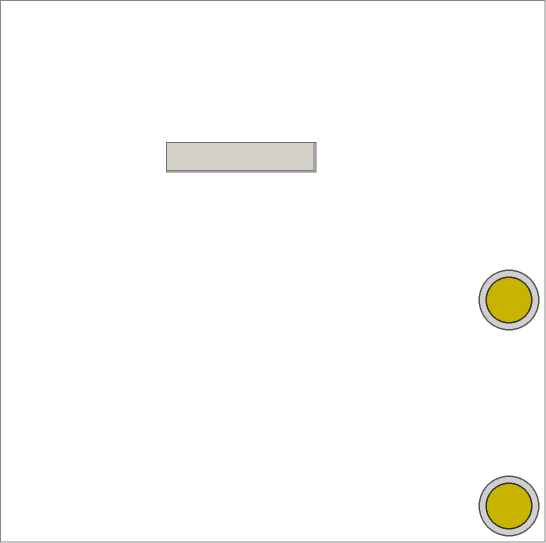
VISUALIZATION Visualization  // 546x543
    Button (166,142 150x30)
        OnMouseClick: toggle MAIN.inputValue
        OnMouseClick: toggle MAIN.inputValue
        OnMouseDown: write MAIN.inputValue via Default
    Lamp1 (474,265 70x70), variable: MAIN.riesingEdge, style: Lamp-Lamp1-Yellow
    Lamp1 (474,471 70x70), variable: MAIN.fallingEdge, style: Lamp-Lamp1-Yellow
END_VISUALIZATION

(* stored: Version 1.1.0.1, ProductVersion 3.1.4022.12
   Visu Visualization: Id {a83dc685-61f1-401e-adc3-fe1b0240dc99} *)
